FUNCTION_BLOCK NumericValue_ID (* Input service interface function block for double word input data *)
  (* Description: Copyright (c) 2017 fortiss GmbH This program and the accompanying materials are made available under the terms of the Eclipse Public License 2.0 which is available at https://www.eclipse.org/legal/epl-2.0/ SPDX-License-Identifier: EPL-2.0 *)
  (* Version 1.0, 2017-03-20, Monika Wenger, fortiss GmbH *)
  PACKAGE isobus::UT::io::NumericValue;
  IMPORT eclipse4diac::core::TypeHash;
  IMPORT isobus::UT::Q::IDs::ID_NULL;
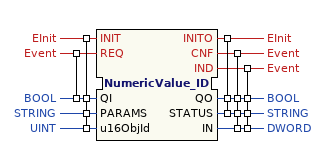
  EVENT_INPUT
    INIT : EInit WITH QI, PARAMS, u16ObjId; (* Service Initialization *)
    REQ WITH QI; (* Service Request *)
  END_EVENT
  EVENT_OUTPUT
    INITO : EInit WITH QO, STATUS; (* Initialization Confirm *)
    CNF WITH QO, STATUS, IN; (* Confirmation of Requested Service *)
    IND WITH QO, STATUS, IN; (* Indication from Resource *)
  END_EVENT
  VAR_INPUT
    QI : BOOL; (* Event Input Qualifier *)
    PARAMS : STRING; (* Service Parameters *)
    u16ObjId : UINT := ID_NULL; (* Object ID *)
  END_VAR
  VAR_OUTPUT
    QO : BOOL; (* Event Output Qualifier *)
    STATUS : STRING; (* Service Status *)
    IN : DWORD; (* Input data from resource *)
  END_VAR
END_FUNCTION_BLOCK
